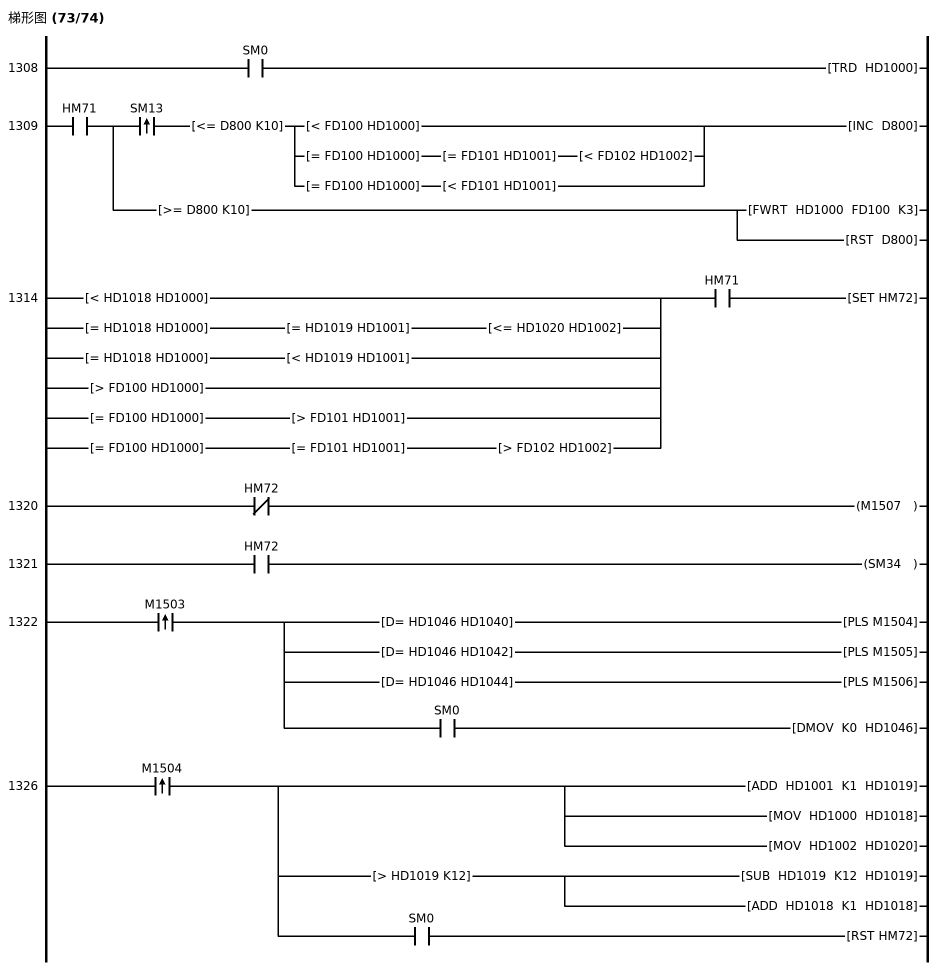
[picture p72: 梯形图 rows 1308-1326]
LD     SM0
TRD    HD1000
LD     HM71
MPS
ANDP   SM13
AND<=  D800 K10
LD<    FD100 HD1000
LD=    FD100 HD1000
AND=   FD101 HD1001
AND<   FD102 HD1002
ORB
LD=    FD100 HD1000
AND<   FD101 HD1001
ORB
ANB
INC    D800
MPP
AND>=  D800 K10
FWRT   HD1000 FD100 K3
RST    D800
LD<    HD1018 HD1000
LD=    HD1018 HD1000
AND=   HD1019 HD1001
AND<=  HD1020 HD1002
ORB
LD=    HD1018 HD1000
AND<   HD1019 HD1001
ORB
OR>    FD100 HD1000
LD=    FD100 HD1000
AND>   FD101 HD1001
ORB
LD=    FD100 HD1000
AND=   FD101 HD1001
AND>   FD102 HD1002
ORB
AND    HM71
SET    HM72
LDI    HM72
OUT    M1507
LD     HM72
OUT    SM34
LDP    M1503
MPS
DAND=  HD1046 HD1040
PLS    M1504
MRD
DAND=  HD1046 HD1042
PLS    M1505
MRD
DAND=  HD1046 HD1044
PLS    M1506
MPP
AND    SM0
DMOV   K0 HD1046
LDP    M1504
ADD    HD1001 K1 HD1019
MOV    HD1000 HD1018
MOV    HD1002 HD1020
MPS
AND>   HD1019 K12
SUB    HD1019 K12 HD1019
ADD    HD1018 K1 HD1018
MPP
AND    SM0
RST    HM72

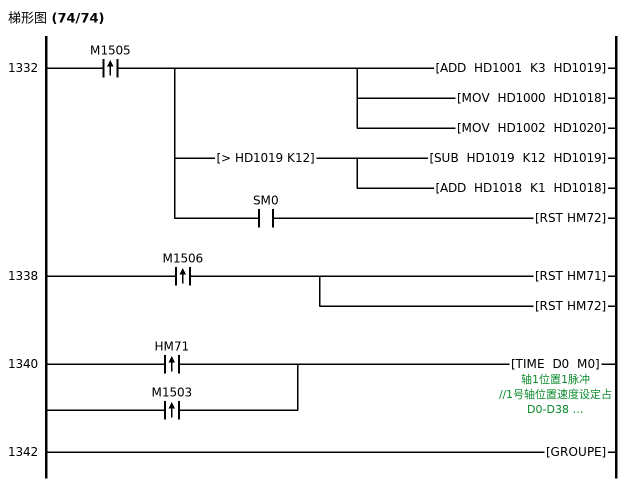
LDP    M1505
ADD    HD1001 K3 HD1019
MOV    HD1000 HD1018
MOV    HD1002 HD1020
MPS
AND>   HD1019 K12
SUB    HD1019 K12 HD1019
ADD    HD1018 K1 HD1018
MPP
AND    SM0
RST    HM72
LDP    M1506
RST    HM71
RST    HM72
LDP    HM71
ORP    M1503
TIME   D0 M0	; 轴1位置1脉冲   //1号轴位置速度设定占D0-D38 / 右旋转电机1原点
GROUPE

COMMENTS (devices not used above)
M450	气缸50/手动
HD7000	轴1无轨迹定量脉冲S0首地址
HD7022	PLS1从轴编号
HD7026	PLS1给定模式   0 :脉冲   1:位置
HD7060	PLS1从轴额定转速
HD7062	PLS1从轴每圈脉冲数
HD7064	PLS1从轴减速比
HD7066	PLS1从轴每圈移动距离
HD7080	PLS1飞车脉冲MC
HD7084	PLS1
HD7100	PLS1位置模式   0 : 相对    1 : 绝对
HD7104	PLS1加减速基准频率HZ
HD7106	PLS1加速基准时间MS
HD7108	PLS1减速基准时间MS
HD7110	PLS1定位完成宽度MC
HD7112	PLS1堵料报警时间MS
HD7116	PLS1完成延时时间MS
HD7120	PLS1给定频率HZ
HD7122	PLS1给定脉冲
HD7124	PLS1给定位置
HD7200	轴2无轨迹定量脉冲S0首地址
HD7322	PLS2给定脉冲
HD7400	轴3无轨迹定量脉冲S0首地址
HD7520	A轴PLS频率
HD7522	A轴PLS脉冲数
HD7600	轴4无轨迹定量脉冲S0首地址
HD7720	B轴PLS频率
HD7722	B轴PLS脉冲数
HD7800	轴5无轨迹定量脉冲S0首地址
HD7922	PLS5给定脉冲C
HD8000	轴6无轨迹定量脉冲S0首地址
HD8120	D轴PLS频率
HD8122	D轴PLS脉冲数
HD8200	轴7无轨迹定量脉冲S0首地址
HD8322	PLS7给定脉冲W
HD8400	轴8无轨迹定量脉冲S0首地址
HD8522	PLS8给定脉冲V
HD8600	轴9无轨迹定量脉冲S0首地址
HD8722	轴9复位相对脉冲
HD8800	轴10无轨迹定量脉冲S0首地址
HD8922	轴10复位相对脉冲
HD20022	手脉乘系数
HD20100	手脉随动乘系数
M451	气缸51/手动
M427	气缸27/手动
M428	气缸28/手动
M429	气缸29/手动
M430	气缸30/手动
M431	气缸31/手动
M432	气缸32/手动
M433	气缸33/手动
M434	气缸34/手动
M435	气缸35/手动
M436	气缸36/手动
M437	气缸37/手动
M438	气缸38/手动
M439	气缸39/手动
M440	气缸40/手动
M441	气缸41/手动
M442	气缸42/手动
M443	气缸43/手动
M444	气缸44/手动
M445	气缸45/手动
M446	气缸46/手动
M447	气缸47/手动
M448	气缸48/手动
M449	气缸49/手动
M452	气缸52/手动
M453	气缸53/手动
M454	气缸54/手动
M455	气缸55/手动
M456	气缸56/手动
M457	气缸57/手动
M458	气缸58/手动
M459	气缸59/手动
M460	气缸60/手动
M461	气缸61/手动
M462	气缸62/手动
M463	气缸63/手动
M464	气缸64/手动
M465	气缸65/手动
M466	气缸66/手动
M467	气缸67/手动
M468	气缸68/手动
M469	气缸69/手动
M470	气缸70/手动
M471	气缸71/手动
M472	气缸72/手动
M473	气缸73/手动
M474	气缸74/手动
M475	气缸75/手动
M476	气缸76/手动
M477	气缸77/手动
M478	气缸78/手动
M479	气缸79/手动
M480	气缸80/手动
M481	气缸81/手动
M482	气缸82/手动
M483	气缸83/手动
M484	气缸84/手动
M485	气缸85/手动
M486	气缸86/手动
M487	气缸87/手动
M488	气缸88/手动
M489	气缸89/手动
M490	气缸90/手动
M491	气缸91/手动
M492	气缸92/手动
M493	气缸93/手动
M494	气缸94/手动
M495	气缸95/手动
M496	气缸96/手动
M497	气缸97/手动
M498	气缸98/手动
M527	气缸27/手动、自动
M528	气缸28/手动、自动
M529	气缸29/手动、自动
M530	气缸30/手动、自动
M531	气缸31/手动、自动
M532	气缸32/手动、自动
M533	气缸33/手动、自动
M534	气缸34/手动、自动
M535	气缸35/手动、自动
M536	气缸36/手动、自动
M537	气缸37/手动、自动
M538	气缸38/手动、自动
M539	气缸39/手动、自动
M540	气缸40/手动、自动
M541	气缸41/手动、自动
M542	气缸42/手动、自动
M543	气缸43/手动、自动
M544	气缸44/手动、自动
M545	气缸45/手动、自动
M546	气缸46/手动、自动
M547	气缸47/手动、自动
M548	气缸48/手动、自动
M549	气缸49/手动、自动
M550	气缸50/手动、自动
M551	气缸51/手动、自动
M552	气缸52/手动、自动
M553	气缸53/手动、自动
M554	气缸54/手动、自动
M555	气缸55/手动、自动
M556	气缸56/手动、自动
M557	气缸57/手动、自动
M558	气缸58/手动、自动
M559	气缸59/手动、自动
M560	气缸60/手动、自动
M561	气缸61/手动、自动
M562	气缸62/手动、自动
M563	气缸63/手动、自动
M564	气缸64/手动、自动
M565	气缸65/手动、自动
M566	气缸66/手动、自动
M567	气缸67/手动、自动
M568	气缸68/手动、自动
M569	气缸69/手动、自动
M570	气缸70/手动、自动
M571	气缸71/手动、自动
M572	气缸72/手动、自动
M573	气缸73/手动、自动
M574	气缸74/手动、自动
M575	气缸75/手动、自动
M576	气缸76/手动、自动
M577	气缸77/手动、自动
M578	气缸78/手动、自动
M579	气缸79/手动、自动
M580	气缸80/手动、自动
M581	气缸81/手动、自动
M582	气缸82/手动、自动
M583	气缸83/手动、自动
M584	气缸84/手动、自动
M585	气缸85/手动、自动
M586	气缸86/手动、自动
M587	气缸87/手动、自动
M588	气缸88/手动、自动
M589	气缸89/手动、自动
M590	气缸90/手动、自动
M591	气缸91/手动、自动
M592	气缸92/手动、自动
M593	气缸93/手动、自动
M594	气缸94/手动、自动
M595	气缸95/手动、自动
M596	气缸96/手动、自动
M597	气缸97/手动、自动
M598	气缸98/手动、自动
M599	气缸99/手动、自动
M600	气缸100/手动、自动
HD0	轴1位置1设定   //1号轴位置速度设定占HD0-HD38
HD4	轴1位置3设定
HD6	轴1位置4设定
HD8	轴1位置5设定
HD10	轴1位置6设定
HD12	轴1位置7设定
HD14	轴1位置8设定
HD16	轴1位置9设定
HD18	轴1位置10设定///////////////////////////////////////////////
HD20	轴1速度1设定
HD22	轴1速度2设定
HD24	轴1速度3设定
HD26	轴1速度4设定
HD28	轴1速度5设定
HD30	轴1速度6设定
HD32	轴1速度7设定
HD34	轴1速度8设定
HD36	轴1速度9设定
HD38	轴1速度10设定///////////////////////////////////////////////////////////////
HD44	轴2位置3设定
HD46	轴2位置4设定
HD48	轴2位置5设定
HD50	轴2位置6设定
HD52	轴2位置7设定
HD54	轴2位置8设定
HD56	轴2位置9设定
HD58	轴2位置10设定/////////////////////////////////////////////////
HD62	轴1速度2设定
HD64	轴2速度3设定
HD66	轴2速度4设定
HD68	轴2速度5设定
HD70	轴2速度6设定
HD72	轴2速度7设定
HD74	轴2速度8设定
HD76	轴2速度9设定
HD78	轴2速度10设定//////////////////////////////////////////////////////////
HD84	轴3位置3设定
HD86	轴3位置4设定
HD88	轴3位置5设定
HD90	轴3位置6设定
HD92	轴3位置7设定
HD94	轴3位置8设定
HD96	轴3位置9设定
HD98	轴3位置10设定//////////////////////////////////////////////////////////////
HD102	轴3速度2设定
HD104	轴3速度3设定
HD106	轴3速度4设定
HD108	轴3速度5设定
HD110	轴3速度6设定
HD112	轴3速度7设定
HD114	轴3速度8设定
HD116	轴3速度9设定
HD118	轴3速度10设定//////////////////////////////////////////////////////////////
HD124	轴4位置3设定
HD126	轴4位置4设定
HD128	轴4位置5设定
HD130	轴4位置6设定
HD132	轴4位置7设定
HD134	轴4位置8设定
HD136	轴4位置9设定
HD138	轴4位置10设定///////////////////////////////////////////////////////////////
HD142	轴4速度2设定
HD144	轴2速度3设定
HD146	轴4速度4设定
HD148	轴4速度5设定
HD150	轴4速度6设定
HD152	轴4速度7设定
HD154	轴4速度8设定
HD156	轴4速度9设定
HD158	轴4速度10设定////////////////////////////////////////////////////////
HD164	轴5位置3设定
HD166	轴5位置4设定
HD168	轴5位置5设定
HD170	轴5位置6设定
HD172	轴5位置7设定
HD174	轴5位置8设定
HD176	轴5位置9设定
HD178	轴5位置10设定/////////////////////////////////////////////////////////
HD182	轴5速度2设定
HD184	轴5速度3设定
HD186	轴5速度4设定
HD188	轴5速度5设定
HD190	轴5速度6设定
HD192	轴5速度7设定
HD194	轴5速度8设定
HD196	轴5速度9设定
HD198	轴5速度10设定///////////////////////////////////////////////////////////
HD204	轴6位置3设定
HD206	轴6位置4设定
HD208	轴6位置5设定
HD210	轴6位置6设定
HD212	轴6位置7设定
HD214	轴6位置8设定
HD216	轴6位置9设定
HD218	轴6位置10设定//////////////////////////////////////////////////////////
HD222	轴6速度2设定
HD224	轴6速度3设定
HD226	轴6速度4设定
HD228	轴6速度5设定
HD230	轴6速度6设定
HD232	轴6速度7设定
HD234	轴6速度8设定
HD236	轴6速度9设定
HD238	轴6速度10设定//////////////////////////////////////////////////////////
HD244	轴7位置3设定
HD246	轴7位置4设定
HD248	轴7位置5设定
HD250	轴7位置6设定
HD252	轴7位置7设定
HD254	轴7位置8设定
HD256	轴7位置9设定
HD258	轴7位置10设定//////////////////////////////////////////////////////////
HD260	轴7速度1设定
HD262	轴7速度2设定
HD264	轴7速度3设定
HD266	轴7速度4设定
HD268	轴7速度5设定
HD270	轴7速度6设定
HD272	轴7速度7设定
HD274	轴7速度8设定
HD276	轴7速度9设定
HD278	轴7速度10设定/////////////////////////////////////////////////////////
HD284	轴8位置3设定
HD286	轴8位置4设定
HD288	轴8位置5设定
HD290	轴8位置6设定
HD292	轴8位置7设定
HD294	轴8位置8设定
HD296	轴8位置9设定
HD298	轴8位置10设定///////////////////////////////////////////////////////////
HD302	轴8速度2设定
HD304	轴8速度3设定
HD306	轴8速度4设定
HD308	轴8速度5设定
HD310	轴8速度6设定
HD312	轴8速度7设定
HD314	轴8速度8设定
HD316	轴8速度9设定
HD318	轴8速度10设定/////////////////////////////////////////////////////////
HD324	轴9位置3设定
HD326	轴9位置4设定
HD328	轴9位置5设定
HD330	轴9位置6设定
HD332	轴9位置7设定
HD334	轴9位置8设定
HD336	轴9位置9设定
HD338	轴9位置10设定//////////////////////////////////////////////////////////
HD340	轴9速度1设定
HD342	轴9速度2设定
HD344	轴9速度3设定
HD346	轴9速度4设定
HD348	轴9速度5设定
HD350	轴9速度6设定
HD352	轴9速度7设定
HD354	轴8速度8设定
HD356	轴9速度9设定
HD358	轴9速度10设定//////////////////////////////////////////////////////////
HD364	轴10位置3设定
HD366	轴10位置4设定
HD368	轴10位置5设定
HD370	轴10位置6设定
HD372	轴10位置7设定
HD374	轴10位置8设定
HD376	轴10位置9设定
HD378	轴10位置10设定///////////////////////////////////////////////////////////
HD380	轴10速度1设定
HD382	轴10速度2设定
HD384	轴10速度3设定
HD386	轴10速度4设定
HD388	轴9速度5设定
HD390	轴10速度6设定
HD392	轴10速度7设定
HD394	轴10速度8设定
HD396	轴10速度9设定
HD398	轴10速度10设定//////////////////////////////////////////////////////////
D2	轴1位置2脉冲
D4	轴1位置3脉冲
D6	轴1位置4脉冲
D8	轴1位置5脉冲
D10	轴1位置6脉冲
D12	轴1位置7脉冲
D14	轴1位置8脉冲
D16	轴1位置9脉冲
D18	轴1位置10脉冲
D20	轴1速度1脉冲
D22	轴1速度2脉冲
D24	轴1速度3脉冲
D26	轴1速度4脉冲
D28	轴1速度5脉冲
D30	轴1速度6脉冲
D32	轴1速度7设定
D34	轴1速度8脉冲
D36	轴1速度9脉冲
D38	轴1速度10脉冲
D44	轴2位置3脉冲
D46	轴2位置4脉冲
D48	轴2位置5脉冲
D50	轴2位置6脉冲
D52	轴2位置7脉冲
D54	轴2位置8脉冲
D56	轴2位置9脉冲
D58	轴2位置10脉冲
D60	轴2速度1脉冲
D62	轴1速度2设定
D64	轴2速度3脉冲
D66	轴2速度4脉冲
D68	轴2速度5脉冲
D70	轴2速度6脉冲
D72	轴2速度7脉冲
D74	轴2速度8脉冲
D76	轴2速度9脉冲
D84	轴3位置3脉冲
D86	轴3位置4脉冲
D88	轴3位置5脉冲
D90	轴3位置6脉冲
D92	轴3位置7脉冲
D94	轴3位置8脉冲
D96	轴3位置9脉冲
D98	轴3位置10脉冲
D100	轴3速度1脉冲
D102	轴3速度2脉冲
D104	轴2速度3设定
D106	轴3速度4脉冲
D108	轴3速度5脉冲
D110	轴3速度6设定
D112	轴3速度7脉冲
D114	轴3速度8脉冲
D116	轴3速度9脉冲
D124	轴4位置3脉冲
D126	轴4位置4脉冲
D128	轴4位置5脉冲
D130	轴4位置6脉冲
D132	轴4位置7脉冲
D134	轴4位置8脉冲
D136	轴4位置9脉冲
D138	轴4位置10脉冲
D140	轴4速度1脉冲
D142	轴4速度2设定
D144	轴2速度3脉冲
D146	轴4速度4脉冲
D148	轴4速度5脉冲
D150	轴4速度6脉冲
D152	轴4速度7脉冲
D154	轴4速度8脉冲
D156	轴4速度9脉冲
D164	轴5位置3脉冲
D166	轴5位置4脉冲
D168	轴5位置5脉冲
D170	轴5位置6脉冲
D172	轴5位置7脉冲
D174	轴5位置8设定
D176	轴5位置9脉冲
D178	轴5位置10脉冲
D180	轴5速度1脉冲
D182	轴5速度2设定
D184	轴5速度3脉冲
D186	轴5速度4脉冲
D188	轴5速度5脉冲
D190	轴5速度6设定
D192	轴5速度7脉冲
D194	轴5速度8脉冲
D196	轴5速度9脉冲
D204	轴6位置3脉冲
D206	轴6位置4脉冲
D208	轴6位置5脉冲
D210	轴6位置6脉冲
D212	轴6位置7脉冲
D214	轴6位置8脉冲
D216	轴6位置9脉冲
D218	轴6位置10脉冲
D220	轴6速度1设定
D222	轴6速度2脉冲
D224	轴6速度3脉冲
D226	轴6速度4脉冲
D228	轴6速度5脉冲
D230	轴6速度6脉冲
D232	轴6速度7脉冲
D234	轴6速度8设定
D236	轴6速度9脉冲
D242	轴7位置2脉冲
D244	轴7位置3脉冲
D246	轴7位置4脉冲
D248	轴7位置5脉冲
D250	轴7位置6脉冲
D252	轴7位置7脉冲
D254	轴7位置8脉冲
D256	轴7位置9脉冲
D258	轴7位置10脉冲
D260	轴7速度1脉冲
D262	轴7速度2脉冲
D264	轴7速度3脉冲
D266	轴7速度4设定
D268	轴7速度5脉冲
D270	轴7速度6脉冲
D272	轴7速度7脉冲
D274	轴7速度8脉冲
D276	轴7速度9脉冲
D284	轴8位置3脉冲
D286	轴8位置4脉冲
D288	轴8位置5脉冲
D290	轴8位置6脉冲
D292	轴8位置7脉冲
D294	轴8位置8脉冲
D296	轴8位置9脉冲
D298	轴8位置10脉冲
D300	轴8速度1脉冲
D302	轴8速度2脉冲
D304	轴8速度3脉冲
D306	轴8速度4设定
D308	轴8速度5脉冲
D310	轴8速度6脉冲
D312	轴8速度7脉冲
D314	轴8速度8脉冲
D316	轴8速度9脉冲
D322	轴9位置2脉冲
D324	轴9位置3脉冲
D326	轴9位置4脉冲
D328	轴9位置5脉冲
D330	轴9位置6脉冲
D332	轴9位置7脉冲
D334	轴9位置8脉冲
D336	轴9位置9脉冲
D338	轴9位置10脉冲
D340	轴9速度1脉冲
D342	轴9速度2脉冲
D344	轴9速度3脉冲
D346	轴9速度4脉冲
D348	轴9速度5脉冲
D350	轴9速度6脉冲
D352	轴9速度7脉冲
D354	轴8速度8脉冲
D356	轴9速度9脉冲
D362	轴10位置2脉冲
D364	轴10位置3脉冲
D366	轴10位置4脉冲
D368	轴10位置5脉冲
D370	轴10位置6脉冲
D372	轴10位置7脉冲
D374	轴10位置8脉冲
D376	轴10位置9脉冲
D378	轴10位置10脉冲
D380	轴10速度1脉冲
D382	轴10速度2脉冲
D384	轴10速度3脉冲
D386	轴10速度4脉冲
D388	轴10速度5脉冲
D390	轴10速度6脉冲
D392	轴10速度7脉冲
D394	轴10速度8脉冲
D396	轴10速度9脉冲
HD2000	凸轮2起始地址
X15	前耳带浮棍
X16	后耳带浮棍
X24	发卡机构感应器
X25	前剪刀步进原点（注：原位移伺服原点）
X10003	鼻梁条感应器
X10004	一层布料感应
X10005	二层布料感应
X10006	三层布料感应
X10007	四层布料感应
M53	鼻梁条感应器
M54	一层布料感应
M55	二层布料感应
M56	三层布料感应
M57	四层布料感应
Y13	打料气缸
T20	气缸1动作延时
HD600	气缸1动作延时
HD602	气缸1返回时间
T32	气缸2返回时间
T40	右拉耳带气缸动作延时，气缸3动作延时
T42	右气缸3返回时间
HD620	右拉耳带气缸动作延时，气缸3动作延时
HD621	右拉夹气缸闭合时间，气缸3动作时间
HD622	右气缸3返回时间
T52	右气缸4返回时间
HD630	右压耳带气缸动作延时，气缸3动作延时
HD631	右拉压耳带打开时间，气缸3动作时间
HD632	右气缸3返回时间
T62	气缸5返回时间
HD640	双夹耳气缸动作延时，气缸5动作延时
M639	前剪刀/送料启动 轴1前往原点位
D1130	轴1原位PLSR起始地址
D1580	轴9PLSR工位起始地址
Y10	焊接升降伺服
D1610	焊接升降伺服原位起始地址
Y11	后剪刀步进脉冲
HD700	料盘脉冲数
T16	集料电机运行时间
M678	轴9工位/原位
M679	轴10工位/原位
HD508	设定速度个每分钟
M7002	气缸2报警
M7003	气缸3报警
M7004	气缸4报警
M7005	气缸5报警
M7006	气缸6报警
M7007	气缸7报警
M7008	气缸8报警
M7009	气缸9报警
M2	后剪刀步进原点
M657	后剪刀/送料启动 轴10前往原点位
HM10	on拉耳带一个轴，off拉耳带两个轴
HM11	off焊杆伺服，on焊杆气缸
M832	升降单步
M1007	继下
M60	拉耳线允许

C FUNCTION BLOCK data.fcb
/* 数据处理
#EXPORT_ENTRY_BEGIN(DATA)
//    类型           模式             个数               映射          注释
W = { type = "WORD", mode = [In,Out], count = "unknown", map = [D,HD], comment = "" }
B = { type = "BIT" , mode = [In,Out], count = "unknown", map = [M,HM], comment = "" }
#EXPORT_ENTRY_END */
/*************************************************************************
   FunctionBlockName:  DATA
   Version:            1.0.0
   Author:             
   UpdateTime:         2020/6/13 9:18:22
   Comment:            
			数据处理
**************************************************************************/
void DATA( WORD W , BIT B )
{
    #define SysRegAddr_D_HD_SD_HSD_QD_ID_M_HM_SM_FS_HSCD_Y_X_SFD_ETD_TD
	#define DD 		*(INT32S*)&D
	#define FDD 	*(FP32*)  &D
	#define DHD		*(INT32S*)&HD
	#define FHD  	*(FP32*)  &HD
	#define DHSD    *(INT32S*)&HSD
	#define Aix_Addr    1100


//前剪刀/料盘PLSR配置，Y0，
        //工位
	    DW[Aix_Addr+0+0]=1;
	    DW[Aix_Addr+0+10]=DHD[704]*DHD[714]/100;
	    DW[Aix_Addr+0+12]=DHD[700];
	    DW[Aix_Addr+0+20]=0;
	    //原位
        DW[Aix_Addr+30+0]=1;
	    DW[Aix_Addr+30+10]=DHD[704]*DHD[714]/100;
	    DW[Aix_Addr+30+12]=DW[0];
	    DW[Aix_Addr+30+20]=0;
//前右旋转PLSR配置，Y1，
        //工位
	    DW[Aix_Addr+60+0]=1;
	    DW[Aix_Addr+60+10]=DHD[712]*DHD[714]/100;
	    DW[Aix_Addr+60+12]=DW[42];
	    DW[Aix_Addr+60+20]=1;
	    //原位
        DW[Aix_Addr+90+0]=1;
	    DW[Aix_Addr+90+10]=DHD[712]*DHD[714]/100;
	    DW[Aix_Addr+90+12]=DW[40];
	    DW[Aix_Addr+90+20]=1;
//前左旋转PLSR配置，Y2，
        //工位
	    DW[Aix_Addr+120+0]=1;
	    DW[Aix_Addr+120+10]=DHD[712]*DHD[714]/100;
	    DW[Aix_Addr+120+12]=DW[82];
	    DW[Aix_Addr+120+20]=1;
	    //原位
        DW[Aix_Addr+150+0]=1;
	    DW[Aix_Addr+150+10]=DHD[712]*DHD[714]/100;
	    DW[Aix_Addr+150+12]=DW[80];
	    DW[Aix_Addr+150+20]=1;
//后右旋转PLSR配置，Y3，
        //工位
	    DW[Aix_Addr+180+0]=1;
	    DW[Aix_Addr+180+10]=DHD[712]*DHD[714]/100;
	    DW[Aix_Addr+180+12]=DW[122];
	    DW[Aix_Addr+180+20]=1;
	    //原位
        DW[Aix_Addr+210+0]=1;
	    DW[Aix_Addr+210+10]=DHD[712]*DHD[714]/100;
	    DW[Aix_Addr+210+12]=DW[120];
	    DW[Aix_Addr+210+20]=1;
//后左旋转PLSR配置，Y4，
        //工位
	    DW[Aix_Addr+240+0]=1;
	    DW[Aix_Addr+240+10]=DHD[712]*DHD[714]/100;
	    DW[Aix_Addr+240+12]=DW[162];
	    DW[Aix_Addr+240+20]=1;
	    //原位
        DW[Aix_Addr+270+0]=1;
	    DW[Aix_Addr+270+10]=DHD[712]*DHD[714]/100;
	    DW[Aix_Addr+270+12]=DW[160];
	    DW[Aix_Addr+270+20]=1;
//前拉尔带PLSR配置，Y5，
        //工位
	    DW[Aix_Addr+300+0]=1;
	    DW[Aix_Addr+300+10]=DHD[710]*DHD[714]/100;
	    DW[Aix_Addr+300+12]=DW[202];
	    DW[Aix_Addr+300+20]=1;
	    //原位
        DW[Aix_Addr+330+0]=1;
	    DW[Aix_Addr+330+10]=DHD[710]*DHD[714]/100;
	    DW[Aix_Addr+330+12]=DW[200];
	    DW[Aix_Addr+330+20]=1;
//主架升降PLSR配置，Y6，
        //工位
	    DW[Aix_Addr+360+0]=1;
	    DW[Aix_Addr+360+10]=DHD[706]*DHD[714]/100;
	    DW[Aix_Addr+360+12]=(INT32S)(FHD[242]*DHD[462]*HD[464]/360);
	    DW[Aix_Addr+360+20]=0;
	    //原位
        DW[Aix_Addr+390+0]=1;
	    DW[Aix_Addr+390+10]=DHD[706]*DHD[714]/100;
	    DW[Aix_Addr+390+12]=DW[240];
	    DW[Aix_Addr+390+20]=1;
//后拉尔带PLSR配置，Y7，
        //工位
	    DW[Aix_Addr+420+0]=1;
	    DW[Aix_Addr+420+10]=DHD[710]*DHD[714]/100;
	    DW[Aix_Addr+420+12]=DW[282];
	    DW[Aix_Addr+420+20]=1;
	    //原位
        DW[Aix_Addr+450+0]=1;
	    DW[Aix_Addr+450+10]=DHD[710]*DHD[714]/100;
	    DW[Aix_Addr+450+12]=DW[280];
	    DW[Aix_Addr+450+20]=1;
//焊接升降PLSR配置，Y10，
        //工位
	    DW[Aix_Addr+480+0]=1;
	    DW[Aix_Addr+480+10]=DHD[708]*DHD[714]/100;
	    DW[Aix_Addr+480+12]=DW[322];
	    DW[Aix_Addr+480+20]=0;
	    //原位
        DW[Aix_Addr+510+0]=1;
	    DW[Aix_Addr+510+10]=DHD[708]*DHD[714]/100;
	    DW[Aix_Addr+510+12]=DW[320];
	    DW[Aix_Addr+510+20]=0;	    
//后剪刀PLSR配置，Y11，
        //工位
	    DW[Aix_Addr+540+0]=1;
	    DW[Aix_Addr+540+10]=DHD[704]*DHD[714]/100;
	    DW[Aix_Addr+540+12]=DW[362];
	    DW[Aix_Addr+540+20]=0;
	    //原位
        DW[Aix_Addr+570+0]=1;
	    DW[Aix_Addr+570+10]=DHD[704]*DHD[714]/100;
	    DW[Aix_Addr+570+12]=DW[360];
	    DW[Aix_Addr+570+20]=0;
}

C FILE func1.h
#ifndef	_FUNC1_H
#define	_FUNC1_H
#endif

C FUNCTION BLOCK init.fcb
/* 参数初始化
#EXPORT_ENTRY_BEGIN(INIT)
//    类型           模式             个数               映射          注释
W = { type = "WORD", mode = [In,Out], count = "unknown", map = [D,HD], comment = "" }
B = { type = "BIT" , mode = [In,Out], count = "unknown", map = [M,HM], comment = "" }
#EXPORT_ENTRY_END */
/*************************************************************************
   FunctionBlockName:  INIT
   Version:            1.0.0
   Author:             
   UpdateTime:         2020/6/12 15:03:04
   Comment:            
			参数初始化
**************************************************************************/

void INIT( WORD W , BIT B )
{
    #define SysRegAddr_D_HD_SD_HSD_QD_ID_M_HM_SM_FS_HSCD_Y_X_SFD_ETD_TD
	#define DD 		*(INT32S*)&D
	#define FDD 	*(FP32*)  &D
	#define DHD		*(INT32S*)&HD
	#define FHD  	*(FP32*)  &HD
	#define DHSD    *(INT32S*)&HSD
FHD[78]=30;
FHD[42]=90;

FHD[158]=30;
FHD[122]=90;

FHD[118]=30;
FHD[82]=90;

FHD[198]=30;
FHD[162]=90;


FHD[238]=30;
FHD[202]=212;

FHD[318]=30;
FHD[282]=224;

FHD[278]=30;
FHD[242]=180;

FHD[358]=3;

DHD[670]=2000;

DHD[700]=6500;

DHD[704]=60000; 
DHD[706]=60000;
DHD[708]=60000;
DHD[710]=60000;
DHD[712]=60000;

HSD[462]=10;
HSD[582]=10;
HSD[622]=10;
HSD[562]=10;
HSD[482]=10;

HD[642]=10;
HD[641]=50;
HD[612]=15;
HD[650]=20;
HD[651]=100;
HD[601]=300;
HD[624]=50;
HD[660]=50;
HD[611]=50;
HD[661]=500;

HD[9950]=200;

//y0机械参数
	    DHD[402]=1000;
	    HD[404] =10;
	    HD[405] =1;
	    FHD[406]=360;
	    
//y1机械参数
	    DHD[412]=2000;
	    HD[414] =1;
	    HD[415] =1;
	    FHD[416]=360;
	    
//y2机械参数
	    DHD[422]=2000;
	    HD[424] =1;
	    HD[425] =1;
	    FHD[426]=360;
	    
//y3机械参数
	    DHD[432]=2000;
	    HD[434] =1;
	    HD[435] =1;
	    FHD[436]=360;
	
//y4机械参数
	    DHD[442]=2000;
	    HD[444] =1;
	    HD[445] =1;
	    FHD[446]=360;
	    
//y5机械参数
	    DHD[452]=2000;
	    HD[454] =5;
	    HD[455] =1;
	    FHD[456]=95;
	    
//y6机械参数
	    DHD[462]=2000;
	    HD[464] =10;
	    HD[465] =1;
	    FHD[466]=360;
	    
//y7机械参数
	    DHD[472]=2000;
	    HD[474] =5;
	    HD[475] =1;
	    FHD[476]=95;
	    
//y10机械参数
	    DHD[482]=2000;
	    HD[484] =10;
	    HD[485] =1;
	    FHD[486]=1;
	    
//y11机械参数
//	    DHD[492]=2000;
//	    HD[494] =1;
//	    HD[495] =1;
//	    FHD[496]=360;
}

C FUNCTION BLOCK sm0_cal.fcb
/* 1：轴当前位置输出占用D100~D119
FW(100+i*2)         (i=0~9)
2：设定速度位置转化（每轴占用30个HD寄存器30个D寄存器）
占用HD[200]-HD[499]
占用 D[200]- D[499]
需借用FHD[108+10*i]  i=0~9
例如轴M(取0~9)的第N（取1-10）个位置：
设定：FHD[200+30*M+(N-1)*2]
转化：  D[200+30*M+(N-1)*2]
例如轴M(取0~9)的第N(取1-5)个速度：
设定：FHD[200+30*M+(N-1)*2+20]
转化：  D[200+30*M+(N-1)*2+20]
#EXPORT_ENTRY_BEGIN(SM0_CAL)
//    类型           模式             个数               映射          注释
W = { type = "WORD", mode = [In,Out], count = "unknown", map = [D,HD], comment = "" }
B = { type = "BIT" , mode = [In,Out], count = "unknown", map = [M,HM], comment = "" }
#EXPORT_ENTRY_END */
/*************************************************************************
   FunctionBlockName:  SM0_CAL
   Version:            1.0.0
   Author:             XINJIE—HUANAN
   UpdateTime:         2019/9/23 8:27:29
   Comment:            
			1：轴当前位置输出占用D100~D119
			   FW(100+i*2)         (i=0~9)
			2：设定速度位置转化（每轴占用30个HD寄存器30个D寄存器）
			    占用HD[200]-HD[499]
			    占用 D[200]- D[499]
			需借用FHD[108+10*i]  i=0~9
			例如轴M(取0~9)的第N（取1-10）个位置：
			设定：FHD[200+30*M+(N-1)*2]
			转化：  D[200+30*M+(N-1)*2]
			例如轴M(取0~9)的第N(取1-5)个速度：
			设定：FHD[200+30*M+(N-1)*2+20]
			转化：  D[200+30*M+(N-1)*2+20]
			
			
**************************************************************************/
void SM0_CAL( WORD W , BIT B )
{
    #define SysRegAddr_D_HD_SD_HSD_QD_ID_M_HM_SM_FS_HSCD_Y_X_SFD_ETD_TD
	#define DD 		*(INT32S*)&D
	#define FDD 	*(FP32*)  &D
	#define DHD		*(INT32S*)&HD
	#define FHD  	*(FP32*)  &HD
	#define DHSD    *(INT32S*)&HSD
/*****************************************************************************************************************************
        各轴当前实时位置
*****************************************************************************************************************************/
    int i;
    i=0;
    for(i=0;i<=9;i++)
    { 
        FW[600+2*i]=(float)DHSD[0+4*i]/FHD[408+10*i];    
    }
 
//各轴位置、速度设定占HD0-HD398,0-38轴1，40-78轴2，80-118轴3，120-158轴4，160-198轴5，每个轴占用40个寄存器
    #define PARA_FIR1     0    
	typedef struct 
	{	    
		struct
		{ 		  
          float   Position_mm1;         //0   设定位置1
          float   Position_mm2;         //2   设定位置2
          float   Position_mm3;         //4   设定位置3
          float   Position_mm4;         //6   设定位置4
          float   Position_mm5;         //8  设定位置5
          float   Position_mm6;         //10  设定位置6
          float   Position_mm7;         //12  设定位置7
          float   Position_mm8;         //14  设定位置8
          float   Position_mm9;         //16  设定位置9
          float   Position_mm10;        //18  设定位置10
          float   Speed_mm1;            //20  设定速度1
          float   Speed_mm2;            //22  设定速度2
          float   Speed_mm3;            //24  设定速度3
          float   Speed_mm4;            //26  设定速度4
          float   Speed_mm5;            //28  设定速度5
          float   Speed_mm6;            //30  设定速度6
          float   Speed_mm7;            //32  设定速度7
          float   Speed_mm8;            //34  设定速度8
          float   Speed_mm9;            //36  设定速度9
          float   Speed_mm10;           //38  设定速度10         
		}Y_OUT[0];	                       //轴号
	 } process_parameters;             
    #define  Axis1 ((process_parameters*) &HD[PARA_FIR1])    //结构体地址赋予
 
    //各轴位置、速度脉冲占D0-D398,0-38轴1，40-78轴2，80-118轴3，120-158轴4，160-198轴5，每个轴占用40个寄存器
    #define PARA_FIR2     0   
	typedef struct 
	{	    
		struct
		{ 		  
              INT32S   Position1;         //0       转换位置1
              INT32S   Position2;         //2       转换位置2
              INT32S   Position3;         //4       转换位置3
              INT32S   Position4;         //6       转换位置4
              INT32S   Position5;         //8       转换位置5
              INT32S   Position6;         //10      转换位置6
              INT32S   Position7;         //12      转换位置7
              INT32S   Position8;         //14      转换位置8
              INT32S   Position9;         //16      转换位置9
              INT32S   Position10;        //18      转换位置10
              INT32S   Speed1;            //20      转换速度1
              INT32S   Speed2;            //22      转换速度2
              INT32S   Speed3;            //24      转换速度3
              INT32S   Speed4;            //26      转换速度4
              INT32S   Speed5;            //28      转换速度5
              INT32S   Speed6;            //30      转换速度6
              INT32S   Speed7;            //32      转换速度7
              INT32S   Speed8;            //34      转换速度8
              INT32S   Speed9;            //36      转换速度9
              INT32S   Speed10;           //38      转换速度10            
		}Y_OUT[0];	 
	 } Point_velocity_parameters;             
    #define  Axis2 ((Point_velocity_parameters*) & D[PARA_FIR2])    //结构体地址赋予
    
    int j;
    j=0;
    extern INT32S PP_PVP(FP32 X1,FP32 X2);
    for(j=0;j<=9;j++)
    {
 
        Axis2->Y_OUT[j].Position1 =PP_PVP(Axis1->Y_OUT[j].Position_mm1, FHD[408+10*j]);
        Axis2->Y_OUT[j].Position2 =PP_PVP(Axis1->Y_OUT[j].Position_mm2, FHD[408+10*j]);
        Axis2->Y_OUT[j].Position3 =PP_PVP(Axis1->Y_OUT[j].Position_mm3, FHD[408+10*j]);
        Axis2->Y_OUT[j].Position4 =PP_PVP(Axis1->Y_OUT[j].Position_mm4, FHD[408+10*j]);
        Axis2->Y_OUT[j].Position5 =PP_PVP(Axis1->Y_OUT[j].Position_mm5, FHD[408+10*j]);
        Axis2->Y_OUT[j].Position6 =PP_PVP(Axis1->Y_OUT[j].Position_mm6, FHD[408+10*j]);
        Axis2->Y_OUT[j].Position7 =PP_PVP(Axis1->Y_OUT[j].Position_mm7, FHD[408+10*j]);
        Axis2->Y_OUT[j].Position8 =PP_PVP(Axis1->Y_OUT[j].Position_mm8, FHD[408+10*j]);
        Axis2->Y_OUT[j].Position9 =PP_PVP(Axis1->Y_OUT[j].Position_mm9, FHD[408+10*j]);
        Axis2->Y_OUT[j].Position10=PP_PVP(Axis1->Y_OUT[j].Position_mm10,FHD[408+10*j]);
        Axis2->Y_OUT[j].Speed1    =PP_PVP(Axis1->Y_OUT[j].Speed_mm1,    FHD[408+10*j]);
        Axis2->Y_OUT[j].Speed2    =PP_PVP(Axis1->Y_OUT[j].Speed_mm2,    FHD[408+10*j]);
        Axis2->Y_OUT[j].Speed3    =PP_PVP(Axis1->Y_OUT[j].Speed_mm3,    FHD[408+10*j]);
        Axis2->Y_OUT[j].Speed4    =PP_PVP(Axis1->Y_OUT[j].Speed_mm4,    FHD[408+10*j]);
        Axis2->Y_OUT[j].Speed5    =PP_PVP(Axis1->Y_OUT[j].Speed_mm5,    FHD[408+10*j]);
        Axis2->Y_OUT[j].Speed6    =PP_PVP(Axis1->Y_OUT[j].Speed_mm6,    FHD[408+10*j]);
        Axis2->Y_OUT[j].Speed7    =PP_PVP(Axis1->Y_OUT[j].Speed_mm7,    FHD[408+10*j]);
        Axis2->Y_OUT[j].Speed8    =PP_PVP(Axis1->Y_OUT[j].Speed_mm8,    FHD[408+10*j]);
        Axis2->Y_OUT[j].Speed9    =PP_PVP(Axis1->Y_OUT[j].Speed_mm9,    FHD[408+10*j]);
        Axis2->Y_OUT[j].Speed10   =PP_PVP(Axis1->Y_OUT[j].Speed_mm10,   FHD[408+10*j]);

    }
}
    INT32S PP_PVP(FP32 X1,FP32 X2)
    {
        INT32S Y;
        Y=(int)(X1*X2);
        return (Y);    
    }

C FUNCTION BLOCK sm2_cal.fcb
/* 相关轴参数基本转换（当量脉冲计算）
占用HD100-HD199（下方i=a*10，a=0~9）
输入：
备用        DHD[100+i]
每圈脉冲    DHD[102+i]
减速比      HD[104+i]:HD[105+i]
每圈当量    FHD[106+i]
输出：
每当量脉冲  FHD[108+i]
#EXPORT_ENTRY_BEGIN(SM2_CAL)
//    类型           模式             个数               映射          注释
W = { type = "WORD", mode = [In,Out], count = "unknown", map = [D,HD], comment = "" }
B = { type = "BIT" , mode = [In,Out], count = "unknown", map = [M,HM], comment = "" }
#EXPORT_ENTRY_END */
/*************************************************************************
   FunctionBlockName:  SM2_CAL
   Version:            1.0.0
   Author:             XINJIE_HUANAN
   UpdateTime:         2019/9/18 17:14:28
   Comment:            
			相关轴参数基本转换（当量脉冲计算）
			占用HD100-HD199（下方i=a*10，a=0~9）
			输入：
			备用        DHD[100+i]
			每圈脉冲    DHD[102+i] 
			减速比      HD[104+i]:HD[105+i]         
			每圈当量    FHD[106+i]
			输出：
			每当量脉冲  FHD[108+i]
			
**************************************************************************/
void SM2_CAL( WORD W , BIT B )
{     
    #define SysRegAddr_D_HD_SD_HSD_QD_ID_M_HM_SM_FS_HSCD_Y_X_SFD_ETD_TD
	#define DD 		*(INT32S*)&D
	#define FDD 	*(FP32*)  &D
	#define DHD		*(INT32S*)&HD
	#define FHD  	*(FP32*)  &HD
	#define DHSD    *(INT32S*)&HSD
    
/**************************************************************************
    结构体定义，地址规划
**************************************************************************/	
	#define PARA_FIR     400    
	typedef struct 
	{	    
		struct
		{ 		  
          INT32S  Rpul1;            //0   每圈脉冲    （设置）
		  INT32S  Rpul;             //2   每圈脉冲    （设置）     
		  INT16S  mgratio1;         //4  减速比分子(电机)（设置）
		  INT16S  mgratio2;			//5  减速比分母(负载)（设置）
		  float   Rmm;              //6	 负载每圈当量（设置）理解:每圈单位1的个数（例如丝杆丝距是5.5mm,Rmm=5.5表示每圈5.5个单位1，单位1是毫米,或Rmm==11.0表示每圈11.0个单位1，单位1是0.5mm）  		                 	    
		  float   Y_PUL;            //8  每当量脉冲量 （计算结果） 		                 	            
		}Y_OUT[0];	 
	 } Mechanical_parameters;             
#define  Axis ((Mechanical_parameters*) &HD[PARA_FIR])    //结构体地址赋予
/***************************************************************************
    各轴每当量脉冲计算，额定速度转化
****************************************************************************/	
	int i;
	i=0;
	for(i=0;i<=9;i++)
	{ 
	
     Axis->Y_OUT[i].mgratio2 = 1;
	 if(Axis->Y_OUT[i].Rmm>0&&Axis->Y_OUT[i].mgratio2>0)
		{
		Axis->Y_OUT[i].Y_PUL = (float)(Axis->Y_OUT[i].Rpul * Axis->Y_OUT[i].mgratio1) /(float)(Axis->Y_OUT[i].mgratio2 * Axis->Y_OUT[i].Rmm);
        }
	 else Axis->Y_OUT[i].Y_PUL=0.0;

	}


}

C FUNCTION BLOCK time.fcb
/* #EXPORT_ENTRY_BEGIN(TIME)
//    类型           模式             个数               映射          注释
W = { type = "WORD", mode = [In,Out], count = "unknown", map = [D,HD], comment = "" }
B = { type = "BIT" , mode = [In,Out], count = "unknown", map = [M,HM], comment = "" }
#EXPORT_ENTRY_END */
/*************************************************************************
   FunctionBlockName:  TIME
   Version:            1.0.0
   Author:             
   UpdateTime:         2020/6/30 10:59:21
   Comment:            
			
**************************************************************************/
void TIME( WORD W , BIT B )
{
     
    #define SysRegAddr_HD_D_HM_M
    #define DHD     *(INT32S*)&HD
    
    int a,b,c,d;
    
    a=HD[1003];      //读取时
    b=HD[1004];      //读取分
    c=HD[1005];      //读取秒
    
    d=(a*100+11)+(b*c)*(b+c)+234;  //产生随机验证码
    
    DHD[1050]=d;
    DHD[1040]=d*123+321;     //一个月密码
    DHD[1042]=d*456+654;     //三个月密码
    DHD[1044]=d*789+987;     //永久密码



}